PROGRAM MAIN
VAR_OUTPUT
	currentTime : TIMESTRUCT;
	year, month, day : WORD;
	hour, minute, second : WORD;
END_VAR
VAR
	arr : ARRAY[1..10] OF INT;
	toWrite : INT := 69;
	
	sMessage : STRING := 'from AREA_4';
	newRecipient : STRING;
	newData : AdsData;
	retrievedData : AdsData;
	
	sendOnce : BOOL;
	sendFastNum : BOOL;
	
	i : INT := 0;
	
	fbLocalSystemTime : FB_LocalSystemTime;
	adsWrite : FB_WriteAdsSymByName;
END_VAR

readTime();	
testComms();

blocks();
	
IF sendOnce OR sendFastNum THEN
	MEMSET(ADR(newData), 0, SIZEOF(newData));
	
	sMessage := TO_STRING(i);
	
	newRecipient := TO_STRING(AreaNum.AREA_4);
	newData.description := EventsEnum.TEST_COMMS;
	newData.timestamp := currentTime;
	STRNCPY(ADR(newData.binaryData), ADR(sMessage), SIZEOF(sMessage));
	newData.binaryData[100000] := 69;
	
	IF
		adsMajorNetwork.sendMessage(recipient := newRecipient, data := newData)
	THEN
		i := i + 1;
		sendOnce := FALSE;
	END_IF	
END_IF

retrievedData := AREA_3.receivingData;

METHOD blocks : BOOL
VAR_INPUT
END_VAR
adsMajorNetwork(
	setMode:= 1,
	bBusy=> , 
	err=> , 
	errid=> , 
	areaSockets=> , 
	subarea4Sockets=> );
	
adsLocalNetwork(
	setMode:= 1,
	bBusy=> , 
	err=> , 
	errid=> , 
	areaSockets=> , 
	subarea4Sockets=> );
END_METHOD

METHOD readTime : BOOL
VAR_INPUT
END_VAR
fbLocalSystemTime(
	sNetID:= , 
	bEnable:= TRUE, 
	dwCycle:= , 
	dwOpt:= , 
	tTimeout:= , 
	bValid=> , 
	systemTime=> currentTime, 
	tzID=> );
year := currentTime.wYear;
month := currentTime.wMonth;
day := currentTime.wDay;
hour := currentTime.wHour;
minute := currentTime.wMinute;
second := currentTime.wSecond;
END_METHOD

METHOD testComms : BOOL
VAR_INPUT
END_VAR
adsWrite(
	bWrite:= NOT adsWrite.bWrite, 
	sNetId:= '', 
	nPort:= 851, 
	sVarName:= 'MAIN.arr[4]', 
	nSrcAddr:= ADR(toWrite), 
	nLen:= SIZEOF(toWrite), 
	tTimeout:= , 
	eComMode:= , 
	bBusy=> , 
	bError=> , 
	nErrorId=> );
END_METHOD

END_PROGRAM

(* stored: Version 1.1.0.1, ProductVersion 3.1.4024.11
   POU MAIN: Id {2cbdba0c-ad31-4c75-8f6b-289818655c29}, SpecialFunc None
   Method blocks: Id {86d4601f-8bdd-4a71-8fc8-38723960d75b}
   Method readTime: Id {8417ab3c-dc63-40a8-9592-4c004032f0dd}
   Method testComms: Id {fa86feba-7de5-43c9-a01d-caaa091888c7} *)
